	FUNCTION_BLOCK FB 104
	TITLE =G004G GENERAL ELEMENTS STEEPING
	//COPYRIGHT:    (C) 2009  BUHLER AG, CH-9240 UZWIL, SWITZERLAND
	//
	//PRODUCT:      WinCoS_BIW01_09
	//
	//TITLE:        GENERAL ELEMENTS STEEPING
	//                General group control
	//                Allgemeine Gruppensteuerung
	//
	//--------------------------------------------------------------------------------
	//
	//IDENT:        AUTHOR:             DEPT:                              DATE:
	//
	//P01_FB104.1.0 K.Renz              CSB41                              13.Jan.2010
	//             1st Release
	//
	//--------------------------------------------------------------------------------
	//
	//PURPOSE:
	//
	//MANUAL :
	//
	//RESTRICTIONS:
	//
	//--------------------------------------------------------------------------------
	AUTHOR  : KR
	FAMILY  : USW
	VERSION : 9.9


	VAR
	  Gr       : FB10;	//Standard interface to group
	  InOutValue1    : DINT; //Data for user
	  InOutValue2    : DINT; //Data for user
	  OutWayConflict : BOOL;	//Data for user
	  OutSelectionOk : BOOL;	//Data for user
	  CmdNewValue : BOOL;	//Data for user
	  CmdNewJob   : BOOL;	//Data for user
	  OutCodeOK   : BOOL;	//Data for user
	  InEndOfJob  : BOOL ;	//Data for user
	  staWayOk      : BOOL ;	//Data for user
	  EdgeStartRelease : BOOL ;	//Data for user
	  USW8  : BOOL;	//Data for user
	  USW9 : BOOL;	//Data for user
	  USW10: BOOL;	//Data for user
	  USW11: BOOL;	//Data for user
	  USW12: BOOL;	//Data for user
	  USW13: BOOL;	//Data for user
	  USW14: BOOL;	//Data for user
	  USW15: BOOL;	//Data for user
	     #A_11_A040Z1 : FB14;   // DigInpCont
	     #A_11_F043Z1 : FB14;   // DigInpCont
	     #A_11_K091Z1 : FB14;   // DigInpCont
	     #A_11_S_H097Z1 : FB14;   // DigInpCont
	     #A_11_A097Z1 : FB14;   // DigInpCont
	     #A_1199_SHE01 : FB14;   // DigInpCont
	     #A_1199_SHE02 : FB14;   // DigInpCont
	END_VAR
	VAR_TEMP
	   tmpEnable		: BOOL;
	   tmpFlag  		: BOOL;
	   tmpCmdNext		: BOOL;
	   tmpLocal  		: BOOL;
	   tmpAspOk  		: BOOL;
	   tmpHWStop 		: BOOL;
	   tmpInstanzDBNo       : INT ;
	END_VAR
	BEGIN
	NETWORK
	TITLE =
	NETWORK
	TITLE =Read command from group control
	//Parameter
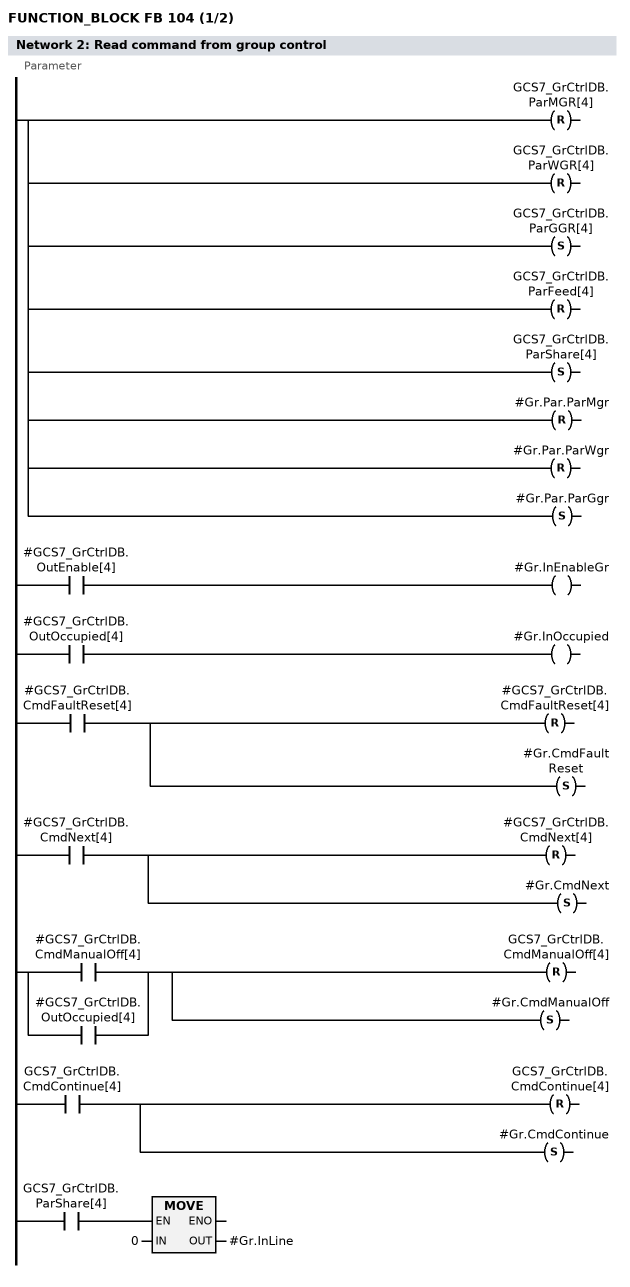
	      SET;
	      R   GCS7_GrCtrlDB.ParMGR[4];
	      R   GCS7_GrCtrlDB.ParWGR[4];
	      S   GCS7_GrCtrlDB.ParGGR[4];
	      R   GCS7_GrCtrlDB.ParFeed[4];
	      S   GCS7_GrCtrlDB.ParShare[4];
	      R   #Gr.Par.ParMgr;
	      R   #Gr.Par.ParWgr;
	      S   #Gr.Par.ParGgr;
	//Command
	      U   #GCS7_GrCtrlDB.OutEnable[4];
	      =   #Gr.InEnableGr;
	      U   #GCS7_GrCtrlDB.OutOccupied[4];
	      =   #Gr.InOccupied;
	      U   #GCS7_GrCtrlDB.CmdFaultReset[4];
	      R   #GCS7_GrCtrlDB.CmdFaultReset[4];
	      S   #Gr.CmdFaultReset;
	      U  #GCS7_GrCtrlDB.CmdNext[4];
	      R   #GCS7_GrCtrlDB.CmdNext[4];
	      S   #Gr.CmdNext;
	      U   #GCS7_GrCtrlDB.CmdManualOff[4];
	      O   #GCS7_GrCtrlDB.OutOccupied[4];
	      R   GCS7_GrCtrlDB.CmdManualOff[4];
	      S   #Gr.CmdManualOff;
	      U  GCS7_GrCtrlDB.CmdContinue[4];
	      R   GCS7_GrCtrlDB.CmdContinue[4];
	      S   #Gr.CmdContinue;
	//Init Line Number
	      U   GCS7_GrCtrlDB.ParShare[4];
	      SPBN WE00;
	      L     0;
	      T     #Gr.InLine;
	WE00: NOP   0;
	NETWORK
	TITLE =Call Methode Control
	// 1. Handle Interface PCControl
	// 2. Prepare mode --> ModePassive,ModeActive,ModeIdling
	// 3. Reset global flags of the group
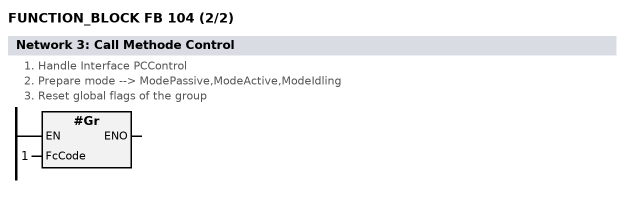
	      CALL #Gr (
	           FcCode                   := 1);
	NETWORK
	TITLE =Restart Idling Time
	      CLR;
	      S    #Gr.CmdRestartIdling;
	NETWORK
	TITLE =Prepare global flags
	NETWORK
	TITLE =Set Pattern (Target position)
	NETWORK
	TITLE =Interlocking WayOk
	//
	NETWORK
	TITLE =Interlocking Autostart
		CLR;
		R   #Gr.OutAutostart;
	NETWORK
	TITLE =Interlocking Enable
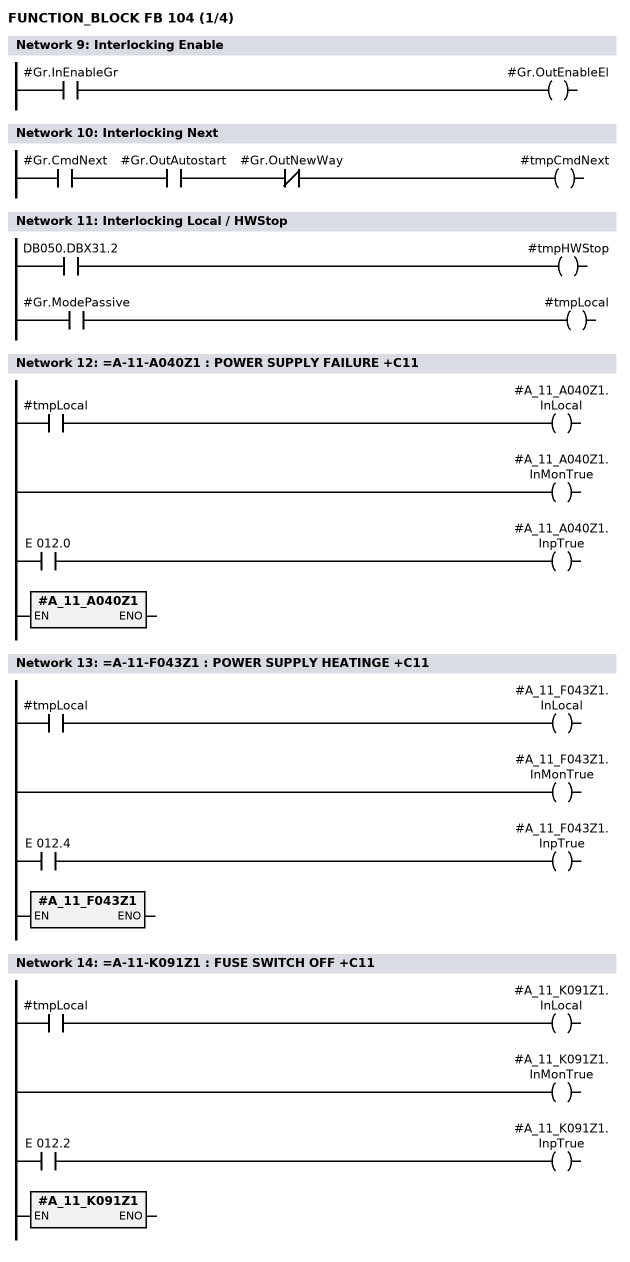
	      U     #Gr.InEnableGr;
	      =     #Gr.OutEnableEl;

	NETWORK
	TITLE =Interlocking Next
	      U     #Gr.CmdNext;
	      U     #Gr.OutAutostart;
	      UN    #Gr.OutNewWay;
	      =    #tmpCmdNext;

	NETWORK
	TITLE =Interlocking Local / HWStop
	      U    DB050.DBX31.2;
	      =    #tmpHWStop;

	      U    #Gr.ModePassive;
	      =    #tmpLocal;

	NETWORK
	TITLE ==A-11-A040Z1 : POWER SUPPLY FAILURE +C11
	NOP 0;
	//-InLocal---
	      U     #tmpLocal;
	      =     #A_11_A040Z1.InLocal;
	//
	//-Monitoring---
	      SET;
	      =      #A_11_A040Z1.InMonTrue;
	//
	//-PreAlarm---
	    //  CLR
	    //  =      #A_11_A040Z1.InPreAlarmTrue
	//
	//-Additional commands---
	//      CLR
	//      S     #A_11_A040Z1.CmdRunTimeOutTime
	//
	//-Read inputs---
	      U     E 012.0;
	      =     #A_11_A040Z1.InpTrue;
	//
	//-Set Parameters---
	//
	//-Call object control---
	      CALL  #A_11_A040Z1;
	//
	//-Write outputs---
	NETWORK
	TITLE ==A-11-F043Z1 : POWER SUPPLY HEATINGE +C11
	NOP 0;
	//-InLocal---
	      U     #tmpLocal;
	      =     #A_11_F043Z1.InLocal;
	//
	//-Monitoring---
	      SET;
	      =      #A_11_F043Z1.InMonTrue;
	//
	//-PreAlarm---
	    //  CLR
	    //  =      #A_11_F043Z1.InPreAlarmTrue
	//
	//-Additional commands---
	//      CLR
	//      S     #A_11_F043Z1.CmdRunTimeOutTime
	//
	//-Read inputs---
	      U     E 012.4;
	      =     #A_11_F043Z1.InpTrue;
	//
	//-Set Parameters---
	//
	//-Call object control---
	      CALL  #A_11_F043Z1;
	//
	//-Write outputs---
	NETWORK
	TITLE ==A-11-K091Z1 : FUSE SWITCH OFF +C11
	NOP 0;
	//-InLocal---
	      U     #tmpLocal;
	      =     #A_11_K091Z1.InLocal;
	//
	//-Monitoring---
	      SET;
	      =      #A_11_K091Z1.InMonTrue;
	//
	//-PreAlarm---
	    //  CLR
	    //  =      #A_11_K091Z1.InPreAlarmTrue
	//
	//-Additional commands---
	//      CLR
	//      S     #A_11_K091Z1.CmdRunTimeOutTime
	//
	//-Read inputs---
	      U     E 012.2;
	      =     #A_11_K091Z1.InpTrue;
	//
	//-Set Parameters---
	//
	//-Call object control---
	      CALL  #A_11_K091Z1;
	//
	//-Write outputs---
	NETWORK
	TITLE ==A-11-S/H097Z1 : OPERATING ON +C11
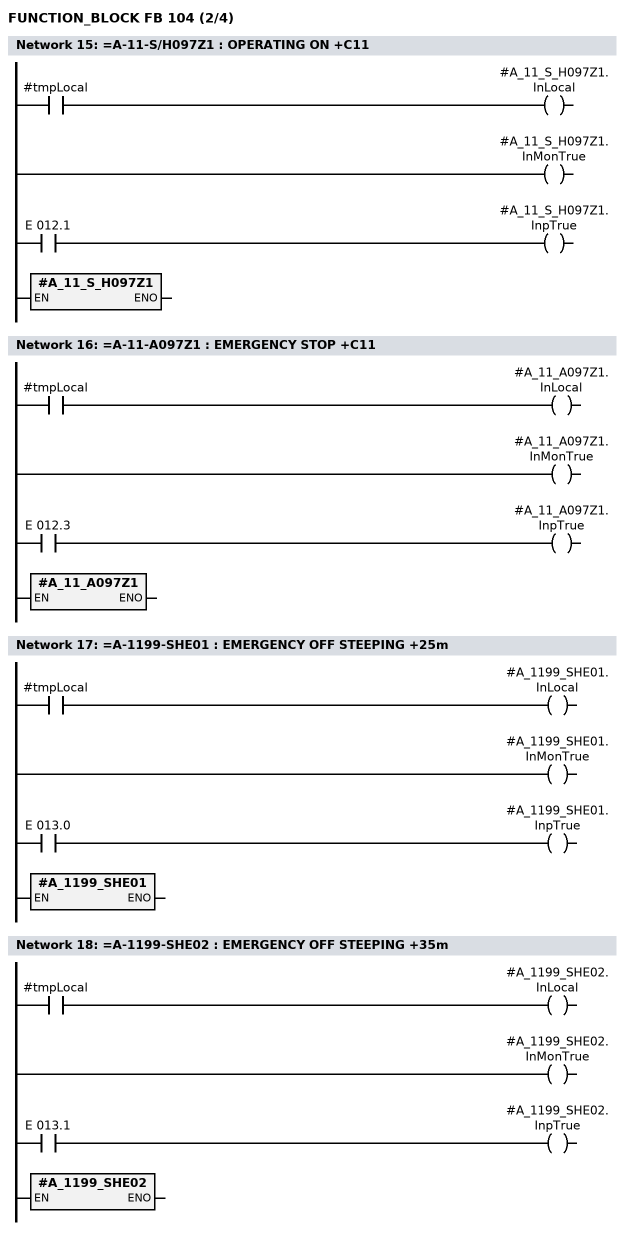
	NOP 0;
	//-InLocal---
	      U     #tmpLocal;
	      =     #A_11_S_H097Z1.InLocal;
	//
	//-Monitoring---
	      SET;
	      =      #A_11_S_H097Z1.InMonTrue;
	//
	//-PreAlarm---
	    //  CLR
	    //  =      #A_11_S_H097Z1.InPreAlarmTrue
	//
	//-Additional commands---
	//      CLR
	//      S     #A_11_S_H097Z1.CmdRunTimeOutTime
	//
	//-Read inputs---
	      U     E 012.1;
	      =     #A_11_S_H097Z1.InpTrue;
	//
	//-Set Parameters---
	//
	//-Call object control---
	      CALL  #A_11_S_H097Z1;
	//
	//-Write outputs---
	NETWORK
	TITLE ==A-11-A097Z1 : EMERGENCY STOP +C11
	NOP 0;
	//-InLocal---
	      U     #tmpLocal;
	      =     #A_11_A097Z1.InLocal;
	//
	//-Monitoring---
	      SET;
	      =      #A_11_A097Z1.InMonTrue;
	//
	//-PreAlarm---
	    //  CLR
	    //  =      #A_11_A097Z1.InPreAlarmTrue
	//
	//-Additional commands---
	//      CLR
	//      S     #A_11_A097Z1.CmdRunTimeOutTime
	//
	//-Read inputs---
	      U     E 012.3;
	      =     #A_11_A097Z1.InpTrue;
	//
	//-Set Parameters---
	//
	//-Call object control---
	      CALL  #A_11_A097Z1;
	//
	//-Write outputs---
	NETWORK
	TITLE ==A-1199-SHE01 : EMERGENCY OFF STEEPING +25m
	NOP 0;
	//-InLocal---
	      U     #tmpLocal;
	      =     #A_1199_SHE01.InLocal;
	//
	//-Monitoring---
	      SET;
	      =      #A_1199_SHE01.InMonTrue;
	//
	//-PreAlarm---
	    //  CLR
	    //  =      #A_1199_SHE01.InPreAlarmTrue
	//
	//-Additional commands---
	//      CLR
	//      S     #A_1199_SHE01.CmdRunTimeOutTime
	//
	//-Read inputs---
	      U     E 013.0;
	      =     #A_1199_SHE01.InpTrue;
	//
	//-Set Parameters---
	//
	//-Call object control---
	      CALL  #A_1199_SHE01;
	//
	//-Write outputs---
	NETWORK
	TITLE ==A-1199-SHE02 : EMERGENCY OFF STEEPING +35m
	NOP 0;
	//-InLocal---
	      U     #tmpLocal;
	      =     #A_1199_SHE02.InLocal;
	//
	//-Monitoring---
	      SET;
	      =      #A_1199_SHE02.InMonTrue;
	//
	//-PreAlarm---
	    //  CLR
	    //  =      #A_1199_SHE02.InPreAlarmTrue
	//
	//-Additional commands---
	//      CLR
	//      S     #A_1199_SHE02.CmdRunTimeOutTime
	//
	//-Read inputs---
	      U     E 013.1;
	      =     #A_1199_SHE02.InpTrue;
	//
	//-Set Parameters---
	//
	//-Call object control---
	      CALL  #A_1199_SHE02;
	//
	//-Write outputs---
	NETWORK
	TITLE =Test Fault
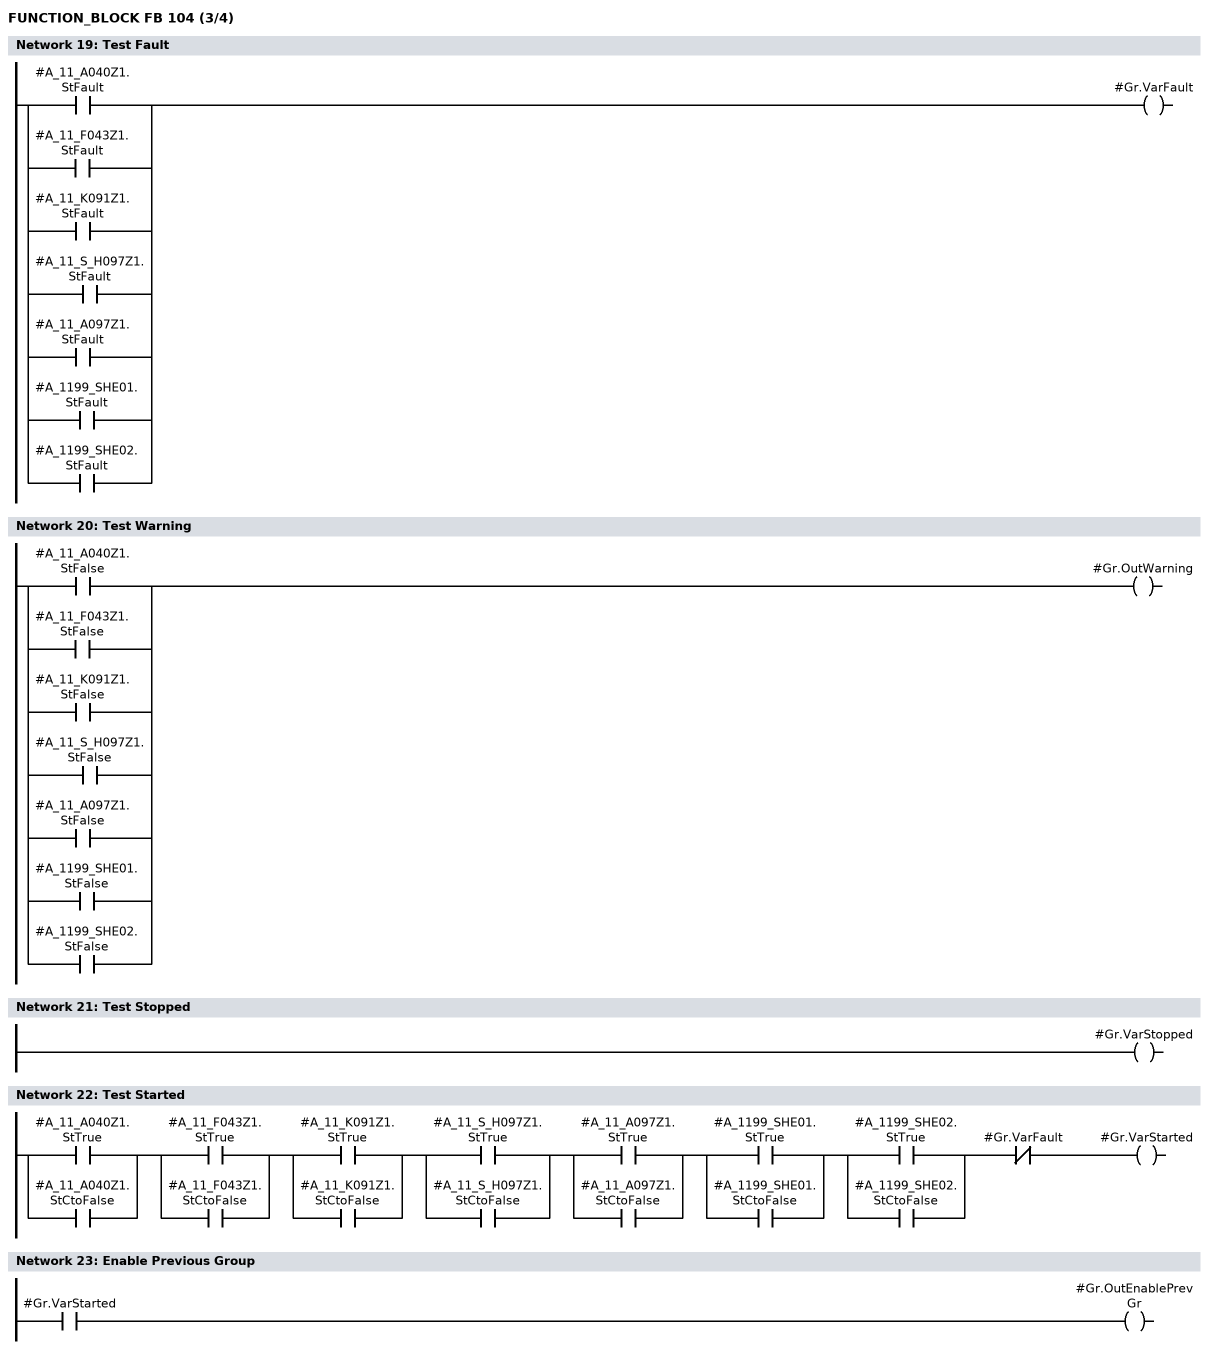
	      U     #A_11_A040Z1.StFault;
	      O     #A_11_F043Z1.StFault;
	      O     #A_11_K091Z1.StFault;
	      O     #A_11_S_H097Z1.StFault;
	      O     #A_11_A097Z1.StFault;
	      O     #A_1199_SHE01.StFault;
	      O     #A_1199_SHE02.StFault;
	      =     #Gr.VarFault;
	NETWORK
	TITLE =Test Warning
	      U     #A_11_A040Z1.StFalse;
	      O     #A_11_F043Z1.StFalse;
	      O     #A_11_K091Z1.StFalse;
	      O     #A_11_S_H097Z1.StFalse;
	      O     #A_11_A097Z1.StFalse;
	      O     #A_1199_SHE01.StFalse;
	      O     #A_1199_SHE02.StFalse;
	      =     #Gr.OutWarning;
	NETWORK
	TITLE =Test Stopped
	      SET;
	      =     #Gr.VarStopped;
	NETWORK
	TITLE =Test Started
	      U(;
	      O     #A_11_A040Z1.StTrue;
	      O     #A_11_A040Z1.StCtoFalse;
	      );
	      U(;
	      O     #A_11_F043Z1.StTrue;
	      O     #A_11_F043Z1.StCtoFalse;
	      );
	      U(;
	      O     #A_11_K091Z1.StTrue;
	      O     #A_11_K091Z1.StCtoFalse;
	      );
	      U(;
	      O     #A_11_S_H097Z1.StTrue;
	      O     #A_11_S_H097Z1.StCtoFalse;
	      );
	      U(;
	      O     #A_11_A097Z1.StTrue;
	      O     #A_11_A097Z1.StCtoFalse;
	      );
	      U(;
	      O     #A_1199_SHE01.StTrue;
	      O     #A_1199_SHE01.StCtoFalse;
	      );
	      U(;
	      O     #A_1199_SHE02.StTrue;
	      O     #A_1199_SHE02.StCtoFalse;
	      );
	      UN  #Gr.VarFault;
	      =     #Gr.VarStarted;
	NETWORK
	TITLE =Enable Previous Group
	      U    #Gr.VarStarted;
	      =     #Gr.OutEnablePrevGr;
	NETWORK
	TITLE =Call Methode State
	//1. Make State of the group: This function use the signals:
	//        Gr.VarStopped, Gr.VarStarted, Gr.VarFault
	//2.Reset Commands to group: e.g.CmdFaultReset
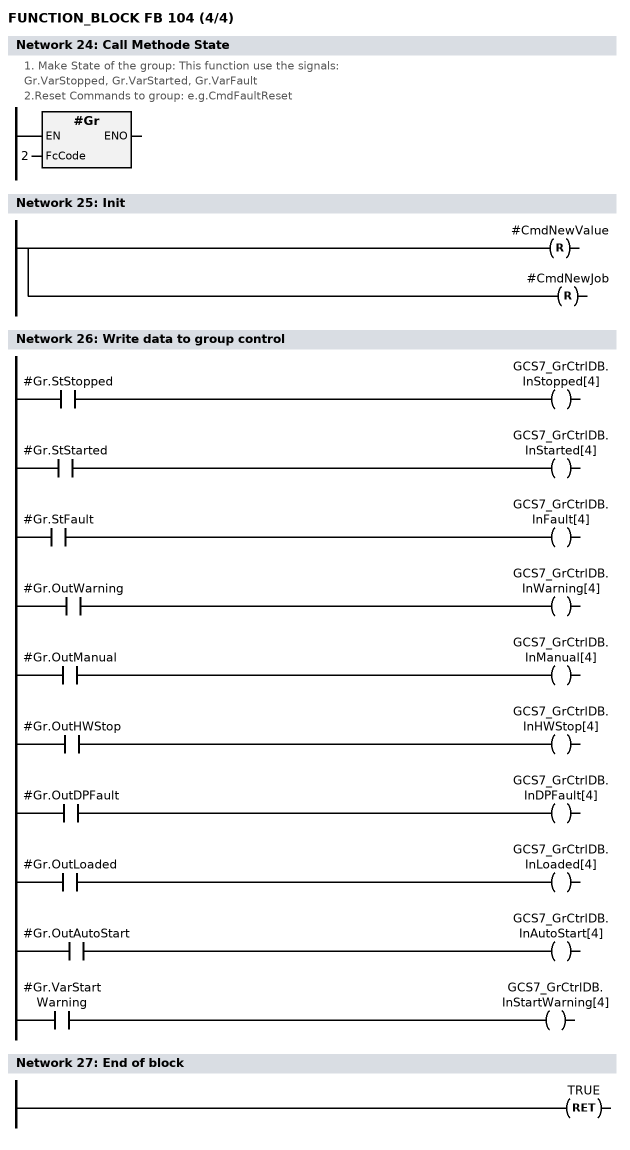
	      CALL #Gr (
	           FcCode                   := 2);
	NETWORK
	TITLE =Init
	      SET;
	      R    #CmdNewValue;
	      R    #CmdNewJob;
	NETWORK
	TITLE =Write data to group control
	      U   #Gr.StStopped;
	      =   GCS7_GrCtrlDB.InStopped[4];
	      U   #Gr.StStarted;
	      =   GCS7_GrCtrlDB.InStarted[4];
	      U   #Gr.StFault;
	      =   GCS7_GrCtrlDB.InFault[4];
	      U   #Gr.OutWarning;
	      =   GCS7_GrCtrlDB.InWarning[4];
	      U   #Gr.OutManual;
	      =   GCS7_GrCtrlDB.InManual[4];
	      U   #Gr.OutHWStop;
	      =   GCS7_GrCtrlDB.InHWStop[4];
	      U   #Gr.OutDPFault;
	      =   GCS7_GrCtrlDB.InDPFault[4];
	      U   #Gr.OutLoaded;
	      =   GCS7_GrCtrlDB.InLoaded[4];
	      U   #Gr.OutAutoStart;
	      =   GCS7_GrCtrlDB.InAutoStart[4];
	      U   #Gr.VarStartWarning;
	      =   GCS7_GrCtrlDB.InStartWarning[4];
	NETWORK
	TITLE =End of block

	BE

	END_FUNCTION_BLOCK
